PROGRAM prgBattery
VAR
	fbBatt						: FB_SunSpec_PV_Inverter_T;
	fbBattCounter				: FB_EnergyCounter;
	lrPowerBatt					: LREAL;						//{#lynus.ag#()}
	dwSOCBattery				: DWORD;						//{#lynus.ag#()}
	byErrorWarningBatt			: BYTE;							//{#lynus.ag#()}
END_VAR
VAR PERSISTENT
	lrCounterBatt				: LREAL;						//{#lynus.ag#()}
END_VAR

// To-Do:
// adopt FB Declaration, change to correct FB
// adopt FB Definition, change to correct in/out Vars
// correct lrPowerBatt definition
// correct lrCounterBatt definition
// correct byErrorWarningBatt definition

fbBatt(
	bEnable:= TRUE, 
	sIPAdress:= '192.168.1.25', 
	byUnitID_Inverter:= 1, 
	stDataSunSpec=> , 
	stDataEMPower_PV=> , 
	stDataEMCounter_PV=> , 
	diNrOfEM_OUT_PV=> );

lrPowerBatt := fbBatt.stDataEMPower_PV.lrPowerTotal;
byErrorWarningBatt := fbBatt.stDataEMPower_PV.byErrorWarning;

fbBattCounter(
	byActiveTariff:= 1, 
	lrPowerInput:= lrPowerBatt, 
	lrTotalCounterEnergy_Consumption=> , 
	lrTotalCounterEnergy_Production=> , 
	lrCounterEnergyT1_Consumption=> , 
	lrCounterEnergyT2_Consumption=> , 
	lrCounterEnergyT1_Production=> , 
	lrCounterEnergyT2_Production=> );
	
IF fbBattCounter.lrTotalCounterEnergy_Consumption > lrCounterBatt THEN  	
	lrCounterBatt := fbBattCounter.lrTotalCounterEnergy_Consumption;
END_IF

END_PROGRAM

(* stored: Version 1.1.0.1, ProductVersion 3.1.4024.11
   POU prgBattery: Id {445907d2-f3d3-45e0-82fc-94f744324500}, SpecialFunc None *)
